{attribute 'qualified_only'}
{attribute 'strict'}
TYPE E_HomeState :
(
	Inactive := 0,
	Jog,
	Delay,
	SetPos,
	P2P,
	HomedReady,
	SecondPhase,
	SecondDelay,
	FinalDelay,
	FinalHoming
);
END_TYPE

(* stored: Version 1.1.0.1, ProductVersion 3.1.4024.12
   DUT E_HomeState: Id {a792deff-22b4-40d6-852c-d8968cabafcd} *)
